TYPE
  (* Standard: 61131-3; Type: Data Type; Description: Table 12, #5 *)
  (* Version 0.1, 2001-03-02, JHC, Rockwell Automation, Tested new Java generation. *)
  (* Version 0.0, 2000-11-09, JHC, Rockwell Automation *)
  (* Compiler header: package fb.rt.ita; *)
  (* Compiler Java IBM VisualAge 3.0 *)
  (* ASN.1 tag PRIVATE 17 *)
  ANALOG_16_INPUT_CONFIGURATION : STRUCT
    SIGNAL_TYPE : ANALOG_SIGNAL_TYPE;
    FILTER : FILTER_PARAMETER;
    CHANNEL : ARRAY [0..15] OF ANALOG_CHANNEL_CONFIGURATION;
  END_STRUCT;
END_TYPE
